// TIA Portal V19 export
TYPE "IFM LMT100_IO"
   STRUCT
      IN : Struct
         Addr : Int;
      END_STRUCT;
      OUT : Struct
         Level : Int;
         Out1 : Bool;
         Out2 : Bool;
      END_STRUCT;
   END_STRUCT;
END_TYPE
